FUNCTION FC_PMCWarningToBoolArray : BOOL
VAR_INPUT
	RegA : POINTER TO BYTE;
END_VAR
VAR_OUTPUT
	WarningList : ARRAY[0..CNC.NUM_MAX_STATION_WARNINGS-1] OF BOOL;
END_VAR
VAR
	i : LWORD;
	j : DINT;
	reg: BYTE;
END_VAR

FOR i:= 0 TO 9 DO
	FOR j := 0 TO 7 DO
        WarningList[(i*8) + j] := TO_BOOL(PBYTE_TO_BYTE((RegA+i)) AND SHL(1,j));
    END_FOR
END_FOR

END_FUNCTION

(* stored: Version 1.1.0.1, ProductVersion 3.1.4024.13
   POU FC_PMCWarningToBoolArray: Id {f9e321ac-8344-4403-85ec-7003d2d69aeb}, SpecialFunc None *)
